Staubli VAL3: onF4Event.pgx

program onF4Event(bool& x_bSave[])
  local bool l_bCheck
  local tool l_tTool
  local string l_sMessage
  local frame l_fNewWorld
begin
  // look if the bButton is enable
  if bButton[3]
    //

      if nIndexTool!=0
        call tcp:checkPoint(l_bCheck)
        if l_bCheck
          call tcp:compose(nIndexTool)
          call tcp:getTool(l_tTool,nIndexTool)
          $jogContext(l_tTool,world,0)
          logMsg("[VALlaser] INTERFACE:Compose the gun")
          x_bSave=true
        else
          call language:message(l_sMessage,122)
          popUpMsg(l_sMessage)
        endIf
      endIf

  endIf
end
